ADAPTER A2X (* unidirectional Adapter Interface for 2 Events and 2 Bools *)
  (* Standard: 61499-1; Description: Copyright (c) 2024 HR Agrartechnik GmbH This program and the accompanying materials are made available under the terms of the Eclipse Public License 2.0 which is available at https://www.eclipse.org/legal/epl-2.0/ SPDX-License-Identifier: EPL-2.0 *)
  (* Version 1.0, 2024-04-24, Franz Höpfinger, HR Agrartechnik GmbH, Initial Version *)
  PACKAGE adapter::types::unidirectional;
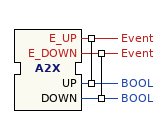
  EVENT_OUTPUT
    E_UP WITH UP; (* UP *)
    E_DOWN WITH DOWN; (* DOWN *)
  END_EVENT
  VAR_OUTPUT
    UP : BOOL; (* TRUE = forward, up, right, clockwise *)
    DOWN : BOOL; (* TRUE = backward, down, left, counter-clockwise *)
  END_VAR
END_ADAPTER
